INTERFACE ITF_CommandChange

METHOD Execute : BOOL
VAR_INPUT
END_VAR
END_METHOD

END_INTERFACE

(* stored: Version 1.1.0.1
   Itf ITF_CommandChange: Id {aec9df3b-b1f6-0d18-0c43-736201fc414a}
   Method Execute: Id {60c49daa-906e-0e4f-1a24-8fb80f45e366} *)
